FUNCTION_BLOCK TcoParentedStructure EXTENDS TcoObject

{attribute 'hide'}
METHOD FB_init : BOOL
VAR_INPUT
	bInitRetains : BOOL; // if TRUE, the retain variables are initialized (warm start / cold start)
	bInCopyCode : BOOL;  // if TRUE, the instance afterwards gets moved into the copy code (online change)
	ParentObject : ITcoObject;	
	ParentStruct : REFERENCE TO TcoStruct;
END_VAR
_Identity := ADR(THIS^);
_ParentObject := ParentObject;
_ParentStruct REF= ParentStruct;
END_METHOD

END_FUNCTION_BLOCK

(* stored: Version 1.1.0.1
   POU TcoParentedStructure: Id {905698ef-b82b-088e-0a1f-f46c1566a649}, SpecialFunc None
   Method FB_init: Id {ed897be3-1063-05a0-051c-b5b35480638d} *)
